FUNCTION_BLOCK WagoSystemWithNetworking (* Composite Function Block Type *)
  (* Standard: 61499-2 *)
  (* Version 0.2, 2003-12-05, JHC, Rockwell Automation, Renamed from NEWCOMPFB. *)
  (* Compiler header: package fb.rt.wago; *)
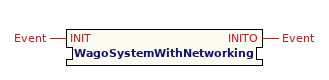
  EVENT_INPUT
    INIT; (* Initialization Request *)
  END_EVENT
  EVENT_OUTPUT
    INITO; (* Initialization Confirm *)
  END_EVENT
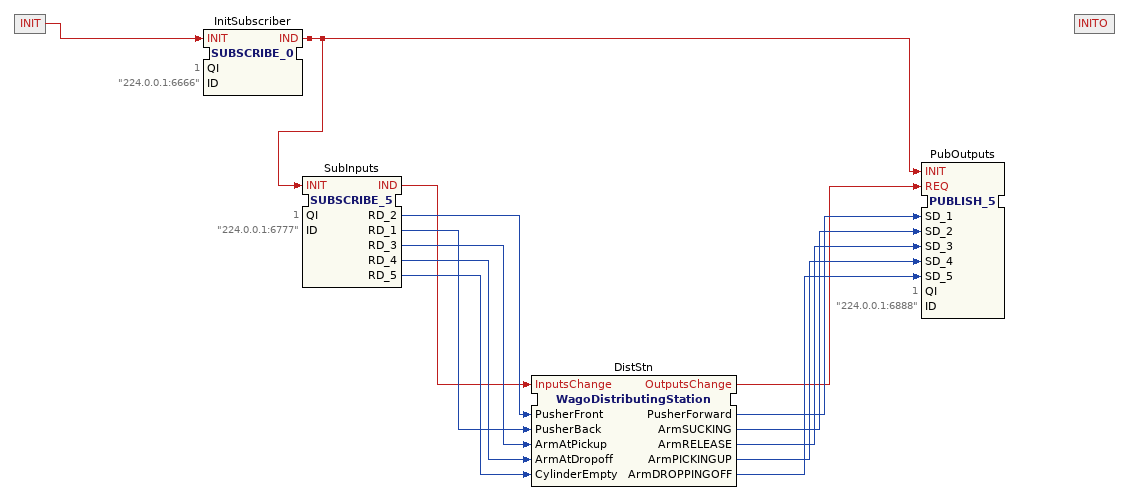
  FBS
    DistStn : WagoDistributingStation;
    SubInputs : SUBSCRIBE_5(QI := 1, ID := "224.0.0.1:6777");
    PubOutputs : PUBLISH_5(QI := 1, ID := "224.0.0.1:6888");
    InitSubscriber : SUBSCRIBE_0(QI := 1, ID := "224.0.0.1:6666");
  END_FBS
  EVENT_CONNECTIONS
    INIT TO InitSubscriber.INIT;
    InitSubscriber.IND TO SubInputs.INIT;
    InitSubscriber.IND TO PubOutputs.INIT;
    SubInputs.IND TO DistStn.InputsChange;
    DistStn.OutputsChange TO PubOutputs.REQ;
  END_CONNECTIONS
  DATA_CONNECTIONS
    SubInputs.RD_2 TO DistStn.PusherFront;
    SubInputs.RD_1 TO DistStn.PusherBack;
    SubInputs.RD_3 TO DistStn.ArmAtPickup;
    SubInputs.RD_4 TO DistStn.ArmAtDropoff;
    SubInputs.RD_5 TO DistStn.CylinderEmpty;
    DistStn.PusherForward TO PubOutputs.SD_1;
    DistStn.ArmSUCKING TO PubOutputs.SD_2;
    DistStn.ArmRELEASE TO PubOutputs.SD_3;
    DistStn.ArmPICKINGUP TO PubOutputs.SD_4;
    DistStn.ArmDROPPINGOFF TO PubOutputs.SD_5;
  END_CONNECTIONS
END_FUNCTION_BLOCK
